# EPICS autosave request: iocBoot/generic_motors_ioc/dbSave/BS_Ps_.req
%
% BURT Request File
%
% $(P)BS:Ps:  Beam Stop Positioner (type: XYZ positioner)
%

file assy.req ASSY=$(P)BS:Ps
file mtr1.req MTR1=$(P)BS:md
file mtr1.req MTR1=$(P)BS:mpt
file mtr1.req MTR1=$(P)BS:myw
file drv1.req DRV1=$(P)BS:D
file drv1.req DRV1=$(P)BS:PT
file drv1.req DRV1=$(P)BS:YW
